FUNCTION_BLOCK overcurrentV2_IO_1_backup (* Composite Function Block Type *)
  (* Standard: 61499-2 *)
  (* Version 0.0, 23/05/2016, Chen-Wei, nxtControl GmbH, template *)
  PACKAGE Main;
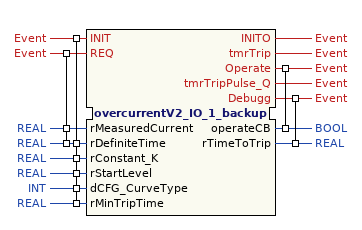
  EVENT_INPUT
    INIT WITH rDefiniteTime, rConstant_K, rStartLevel, dCFG_CurveType, rMinTripTime; (* Initialization Request *)
    REQ WITH rMeasuredCurrent, rDefiniteTime; (* Normal Execution Request *)
  END_EVENT
  EVENT_OUTPUT
    INITO; (* Initialization Confirm *)
    tmrTrip; (* Execution Confirmation *)
    Operate WITH operateCB; (* Delayed Event *)
    tmrTripPulse_Q; (* Delayed Event *)
    Debugg WITH rTimeToTrip;
  END_EVENT
  VAR_INPUT
    rMeasuredCurrent : REAL; (* Input event qualifier *)
    rDefiniteTime : REAL;
    rConstant_K : REAL;
    rStartLevel : REAL;
    dCFG_CurveType : INT;
    rMinTripTime : REAL;
  END_VAR
  VAR_OUTPUT
    operateCB : BOOL; (* Output event qualifier *)
    rTimeToTrip : REAL;
  END_VAR
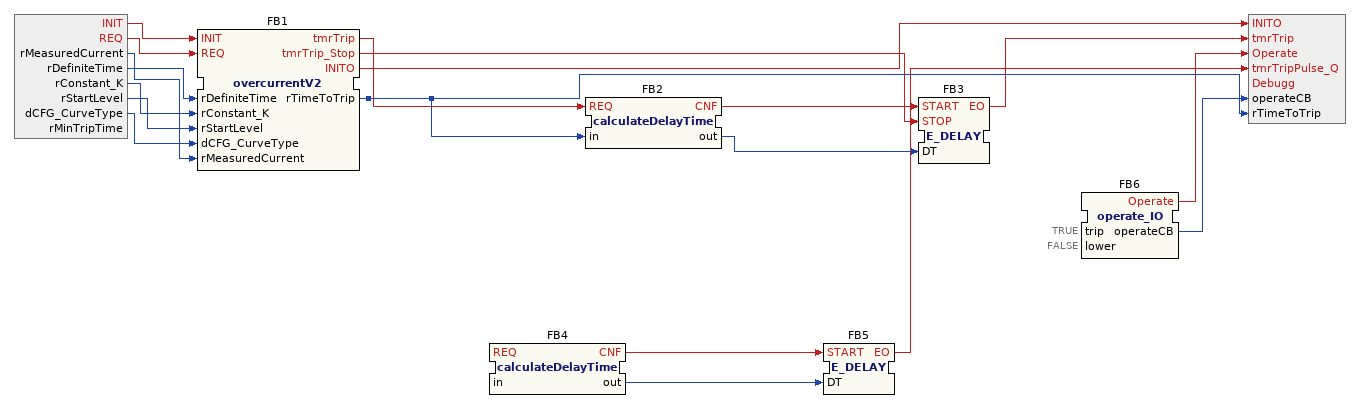
  FBS
    FB2 : calculateDelayTime;
    FB3 : E_DELAY;
    FB4 : calculateDelayTime;
    FB5 : E_DELAY;
    FB6 : operate_IO(trip := TRUE, lower := FALSE);
    FB1 : overcurrentV2;
  END_FBS
  EVENT_CONNECTIONS
    INIT TO FB1.INIT;
    FB2.CNF TO FB3.START;
    FB1.tmrTrip TO FB2.REQ;
    FB3.EO TO tmrTrip;
    FB6.Operate TO Operate;
    REQ TO FB1.REQ;
    FB4.CNF TO FB5.START;
    FB5.EO TO tmrTripPulse_Q;
    FB1.tmrTrip_Stop TO FB3.STOP;
    FB1.INITO TO INITO;
  END_CONNECTIONS
  DATA_CONNECTIONS
    FB2.out TO FB3.DT;
    FB1.rTimeToTrip TO FB2.in;
    FB6.operateCB TO operateCB;
    rDefiniteTime TO FB1.rDefiniteTime;
    rConstant_K TO FB1.rConstant_K;
    rStartLevel TO FB1.rStartLevel;
    dCFG_CurveType TO FB1.dCFG_CurveType;
    rMeasuredCurrent TO FB1.rMeasuredCurrent;
    FB4.out TO FB5.DT;
    FB1.rTimeToTrip TO rTimeToTrip;
  END_CONNECTIONS
END_FUNCTION_BLOCK
